(* LS Electric XG5000 project: XMC_E16A_ModTCP_Client *)
(* PLC LSPLC *)
(* module base 0 slot 0: Input/Output Module:XMC-DN24 (DC 24V Input 8Points/TR output 16Points) *)
(* module base 0 slot 1: Internal Analog Input/Output:XMF-AH04E (A/D voltage/current 2 channels, D/A voltage 2 channels) *)
(* task Periodic Task: Kind=2 *)
(* task Initialization Task: Kind=1 *)
(* task NC Program: Kind=6 *)

PROGRAM ModTCP_Read_FBs (* task: Scan Program *)
(* program showing examples of reading data from a Mod TCP server *)
VAR
    doFC1 : BOOL;
    doFC2 : BOOL;
    doFC3 : BOOL;
    doFC4 : BOOL; (* run function code 4 fb *)
    ErrorCount : INT;
    FC1 : MODBUS_READ_COILS_FC01; (* function code 1 fb *)
    fc1Data : ARRAY[0..1999] OF BOOL;
    FC1_UnitID : USINT; (* UnitID for FC1 fb *)
    FC2 : MODBUS_READ_DISCRETE_INPUTS_FC02; (* function code 2 fb *)
    fc2Data : ARRAY[0..1999] OF BOOL;
    FC2_UnitID : USINT; (* UnitID for FC2 fb *)
    FC3 : MODBUS_READ_HOLDING_REGISTER_FC03; (* function code 3 fb *)
    fc3Data : ARRAY[0..124] OF UINT;
    FC3_UnitID : USINT; (* UnitID for FC3 fb *)
    FC4 : MODBUS_READ_INPUT_REGISTERS_FC04; (* function code 4 fb *)
    fc4Data : ARRAY[0..124] OF UINT; (* data for function code 4 *)
    FC4_UnitID : USINT; (* UnitID for FC4 fb *)
    ipAddr : ARRAY[0..3] OF USINT;
    NonSocketError : BOOL;
    ResetDelay1 : TMR;
    ResetDelay2 : TMR;
    ResetDelay3 : TMR;
    SocketError : BOOL;
    StartResDelay1 : BOOL;
    StartResDelay2 : BOOL;
    STRFindIndex : INT;
    TCP_CheckSock1 : SOCKET_SVCINFO;
    TCP_CheckState1 : BOOL;
    TCP_Close1 : BOOL;
    TCP_Connect1 : BOOL;
    TCP_Sock1 : SOCKET_TCPCONNECT;
    TCP_SockClose : SOCKET_CLOSE;
END_VAR
VAR
    _p1 : BOOL;
END_VAR

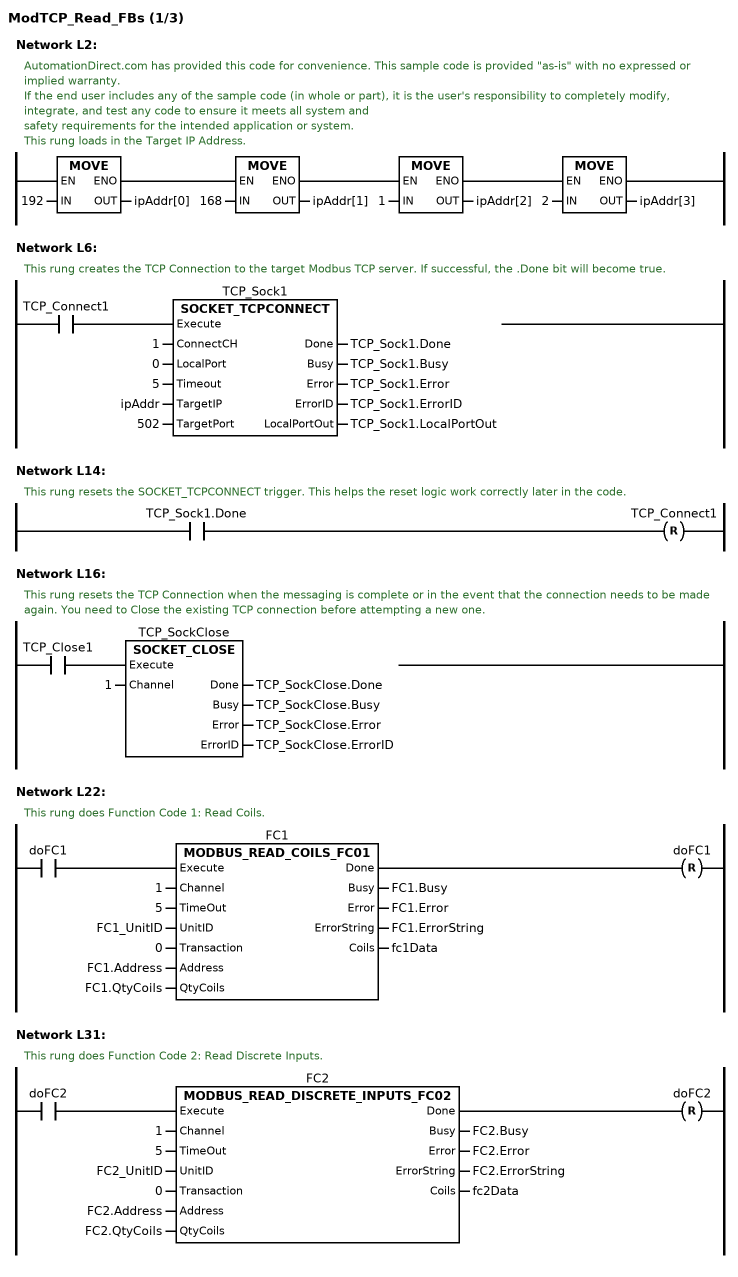
(* AutomationDirect.com has provided this code for convenience. This sample code is provided "as-is" with no expressed or implied warranty. / If the end user includes any of the sample code (in whole or part), it is the user's responsibility to completely modify, integrate, and test any code to ensure it meets all system and / safety requirements for the intended application or system. *)
(* This rung loads in the Target IP Address. *)
(* Rung L2 *)
ipAddr[0] := 192;
ipAddr[1] := 168;
ipAddr[2] := 1;
ipAddr[3] := 2;
(* This rung creates the TCP Connection to the target Modbus TCP server. If successful, the .Done bit will become true. *)
(* Rung L6 *)
TCP_Sock1(Execute := TCP_Connect1, ConnectCH := 1, LocalPort := 0, Timeout := 5, TargetIP := ipAddr, TargetPort := 502, Done => TCP_Sock1.Done, Busy => TCP_Sock1.Busy, Error => TCP_Sock1.Error, ErrorID => TCP_Sock1.ErrorID, LocalPortOut => TCP_Sock1.LocalPortOut);
(* This rung resets the SOCKET_TCPCONNECT trigger. This helps the reset logic work correctly later in the code. *)
(* Rung L14 *)
IF TCP_Sock1.Done THEN TCP_Connect1 := FALSE; END_IF;
(* This rung resets the TCP Connection when the messaging is complete or in the event that the connection needs to be made again. You need to Close the existing TCP connection before attempting a new one. *)
(* Rung L16 *)
TCP_SockClose(Execute := TCP_Close1, Channel := 1, Done => TCP_SockClose.Done, Busy => TCP_SockClose.Busy, Error => TCP_SockClose.Error, ErrorID => TCP_SockClose.ErrorID);
(* This rung does Function Code 1: Read Coils. *)
(* Rung L22 *)
FC1(Execute := doFC1, Channel := 1, TimeOut := 5, UnitID := FC1_UnitID, Transaction := 0, Address := FC1.Address, QtyCoils := FC1.QtyCoils, Busy => FC1.Busy, Error => FC1.Error, ErrorString => FC1.ErrorString, Coils => fc1Data);
IF FC1.Done THEN doFC1 := FALSE; END_IF;
(* This rung does Function Code 2: Read Discrete Inputs. *)
(* Rung L31 *)
FC2(Execute := doFC2, Channel := 1, TimeOut := 5, UnitID := FC2_UnitID, Transaction := 0, Address := FC2.Address, QtyCoils := FC2.QtyCoils, Busy => FC2.Busy, Error => FC2.Error, ErrorString => FC2.ErrorString, Coils => fc2Data);
IF FC2.Done THEN doFC2 := FALSE; END_IF;

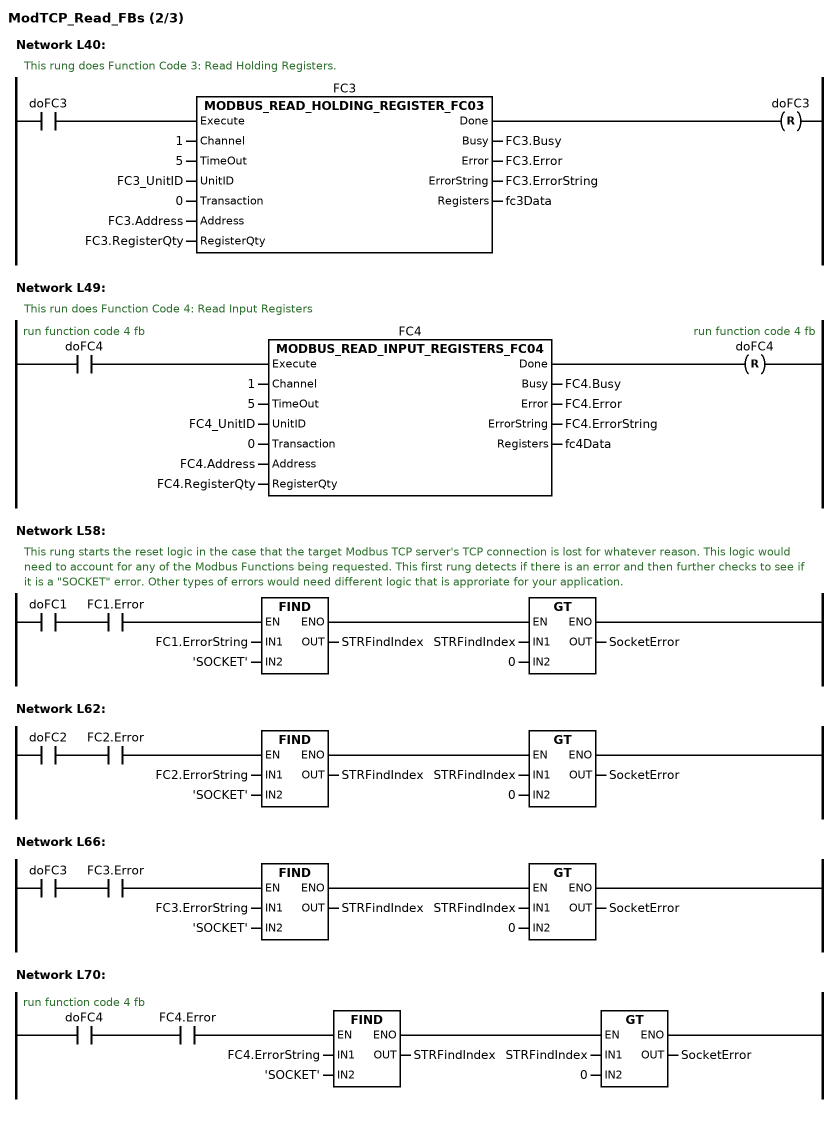
(* This rung does Function Code 3: Read Holding Registers. *)
(* Rung L40 *)
FC3(Execute := doFC3, Channel := 1, TimeOut := 5, UnitID := FC3_UnitID, Transaction := 0, Address := FC3.Address, RegisterQty := FC3.RegisterQty, Busy => FC3.Busy, Error => FC3.Error, ErrorString => FC3.ErrorString, Registers => fc3Data);
IF FC3.Done THEN doFC3 := FALSE; END_IF;
(* This run does Function Code 4: Read Input Registers *)
(* Rung L49 *)
FC4(Execute := doFC4, Channel := 1, TimeOut := 5, UnitID := FC4_UnitID, Transaction := 0, Address := FC4.Address, RegisterQty := FC4.RegisterQty, Busy => FC4.Busy, Error => FC4.Error, ErrorString => FC4.ErrorString, Registers => fc4Data);
IF FC4.Done THEN doFC4 := FALSE; END_IF;
(* This rung starts the reset logic in the case that the target Modbus TCP server's TCP connection is lost for whatever reason. This logic would need to account for any of the Modbus Functions being requested. This first rung detects if there is an error and then further checks to see if it is a "SOCKET" error. Other types of errors would need different logic that is approriate for your application. *)
(* Rung L58 *)
IF doFC1 AND FC1.Error THEN
    STRFindIndex := FIND(FC1.ErrorString, 'SOCKET');
    SocketError := STRFindIndex > 0;
END_IF;
(* Rung L62 *)
IF doFC2 AND FC2.Error THEN
    STRFindIndex := FIND(FC2.ErrorString, 'SOCKET');
    SocketError := STRFindIndex > 0;
END_IF;
(* Rung L66 *)
IF doFC3 AND FC3.Error THEN
    STRFindIndex := FIND(FC3.ErrorString, 'SOCKET');
    SocketError := STRFindIndex > 0;
END_IF;
(* Rung L70 *)
IF doFC4 AND FC4.Error THEN
    STRFindIndex := FIND(FC4.ErrorString, 'SOCKET');
    SocketError := STRFindIndex > 0;
END_IF;

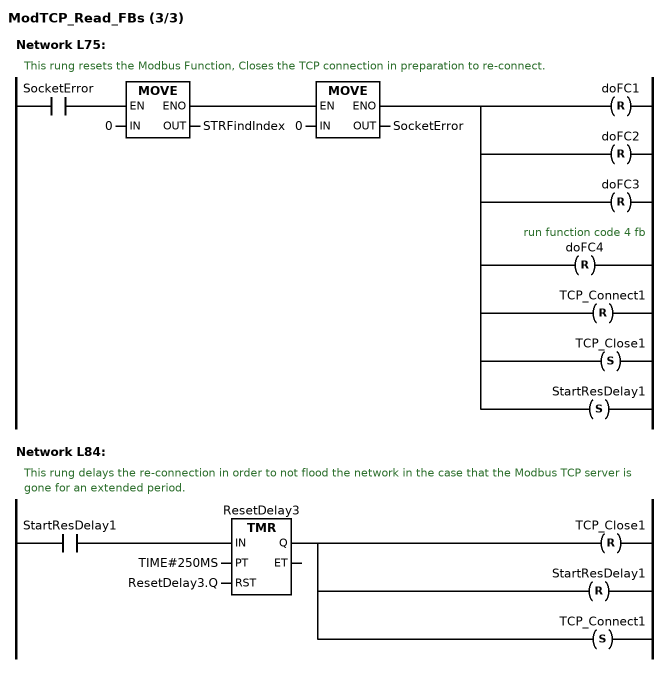
(* This rung resets the Modbus Function, Closes the TCP connection in preparation to re-connect. *)
(* Rung L75 *)
IF SocketError THEN STRFindIndex := 0; END_IF;
_p1 := SocketError;
IF _p1 THEN
    SocketError := 0;
    doFC1 := FALSE;
    doFC2 := FALSE;
    doFC3 := FALSE;
    doFC4 := FALSE;
    TCP_Connect1 := FALSE;
    TCP_Close1 := TRUE;
    StartResDelay1 := TRUE;
END_IF;
(* This rung delays the re-connection in order to not flood the network in the case that the Modbus TCP server is gone for an extended period. *)
(* Rung L84 *)
ResetDelay3(IN := StartResDelay1, PT := TIME#250MS, RST := ResetDelay3.Q);
IF ResetDelay3.Q THEN
    TCP_Close1 := FALSE;
    StartResDelay1 := FALSE;
    TCP_Connect1 := TRUE;
END_IF;
END_PROGRAM

PROGRAM ModTCP_Write_FBs (* task: Scan Program *)
(* example of ModBus TCP Write function blocks *)
VAR
    doFC15 : BOOL; (* execute function code 15 *)
    doFC16 : BOOL; (* execute function code 16 *)
    doFC5 : BOOL; (* execute function code 5 fb *)
    doFC6 : BOOL; (* execute function code 6 *)
    FC15 : MODBUS_WRITE_MULTIPLE_COILS_FC15; (* fb for function code 15 *)
    FC15_data : ARRAY[0..1967] OF BOOL;
    FC15_UnitID : USINT;
    FC16 : MODBUS_WRITE_MULTIPLE_REGISTERS_FC16; (* fb for function code 16 *)
    FC16_data : ARRAY[0..122] OF UINT;
    FC16_UnitID : USINT;
    FC5 : MODBUS_WRITE_SINGLE_COIL_FC05; (* function code 5 fb *)
    FC5_data : BOOL; (* data for fc5 *)
    FC5_UnitID : USINT;
    FC6 : MODBUS_WRITE_SINGLE_REGISTER_FC06; (* fb for function code 6 *)
    FC6_data : UINT;
    FC6_UnitID : USINT;
    ipAddr : ARRAY[0..3] OF USINT;
    ResetDelay3 : TMR;
    SocketError : BOOL;
    StartResDelay1 : BOOL;
    STRFindIndex : INT;
    TCP_Close1 : BOOL;
    TCP_Connect1 : BOOL;
    TCP_Sock1 : SOCKET_TCPCONNECT;
    TCP_SockClose : SOCKET_CLOSE;
END_VAR
VAR
    _p1 : BOOL;
END_VAR

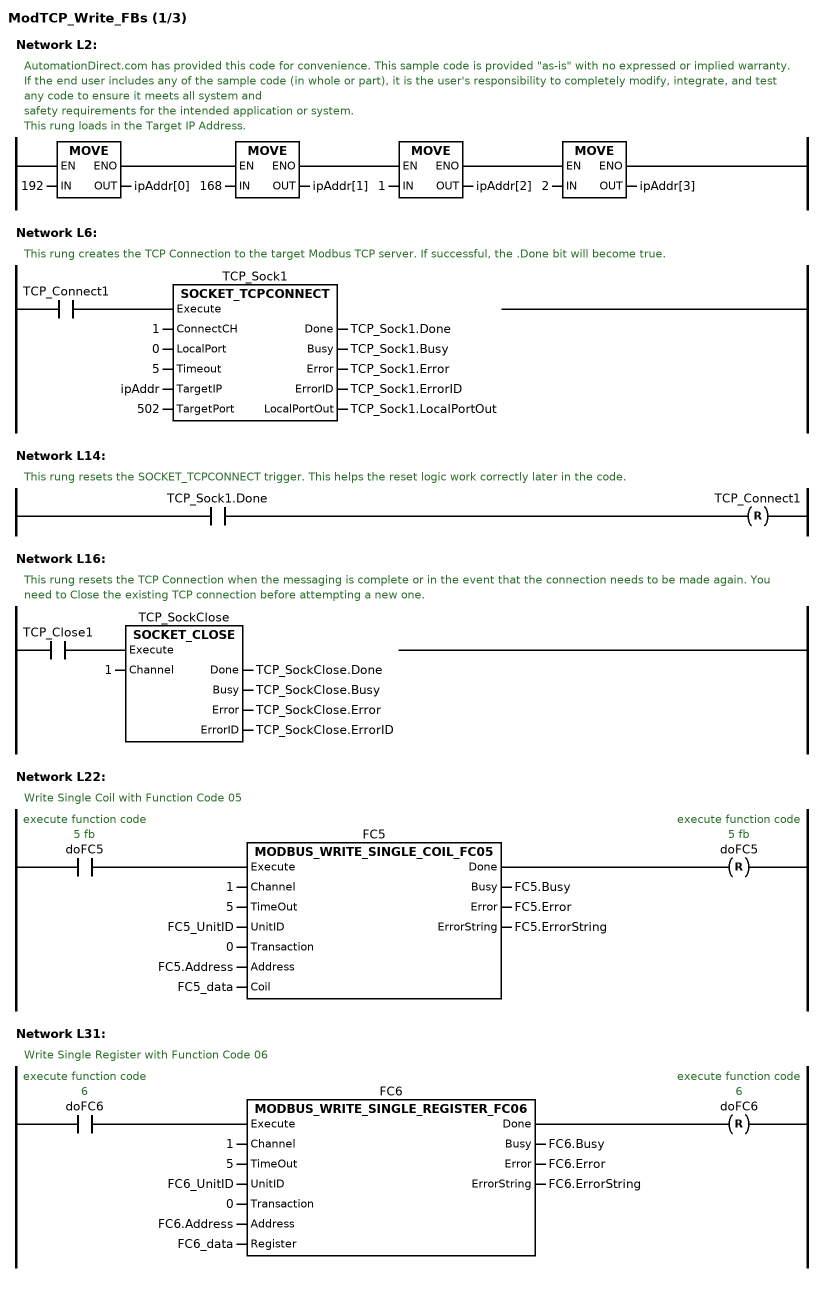
(* AutomationDirect.com has provided this code for convenience. This sample code is provided "as-is" with no expressed or implied warranty. / If the end user includes any of the sample code (in whole or part), it is the user's responsibility to completely modify, integrate, and test any code to ensure it meets all system and / safety requirements for the intended application or system. *)
(* This rung loads in the Target IP Address. *)
(* Rung L2 *)
ipAddr[0] := 192;
ipAddr[1] := 168;
ipAddr[2] := 1;
ipAddr[3] := 2;
(* This rung creates the TCP Connection to the target Modbus TCP server. If successful, the .Done bit will become true. *)
(* Rung L6 *)
TCP_Sock1(Execute := TCP_Connect1, ConnectCH := 1, LocalPort := 0, Timeout := 5, TargetIP := ipAddr, TargetPort := 502, Done => TCP_Sock1.Done, Busy => TCP_Sock1.Busy, Error => TCP_Sock1.Error, ErrorID => TCP_Sock1.ErrorID, LocalPortOut => TCP_Sock1.LocalPortOut);
(* This rung resets the SOCKET_TCPCONNECT trigger. This helps the reset logic work correctly later in the code. *)
(* Rung L14 *)
IF TCP_Sock1.Done THEN TCP_Connect1 := FALSE; END_IF;
(* This rung resets the TCP Connection when the messaging is complete or in the event that the connection needs to be made again. You need to Close the existing TCP connection before attempting a new one. *)
(* Rung L16 *)
TCP_SockClose(Execute := TCP_Close1, Channel := 1, Done => TCP_SockClose.Done, Busy => TCP_SockClose.Busy, Error => TCP_SockClose.Error, ErrorID => TCP_SockClose.ErrorID);
(* Write Single Coil with Function Code 05 *)
(* Rung L22 *)
FC5(Execute := doFC5, Channel := 1, TimeOut := 5, UnitID := FC5_UnitID, Transaction := 0, Address := FC5.Address, Coil := FC5_data, Busy => FC5.Busy, Error => FC5.Error, ErrorString => FC5.ErrorString);
IF FC5.Done THEN doFC5 := FALSE; END_IF;
(* Write Single Register with Function Code 06 *)
(* Rung L31 *)
FC6(Execute := doFC6, Channel := 1, TimeOut := 5, UnitID := FC6_UnitID, Transaction := 0, Address := FC6.Address, Register := FC6_data, Busy => FC6.Busy, Error => FC6.Error, ErrorString => FC6.ErrorString);
IF FC6.Done THEN doFC6 := FALSE; END_IF;

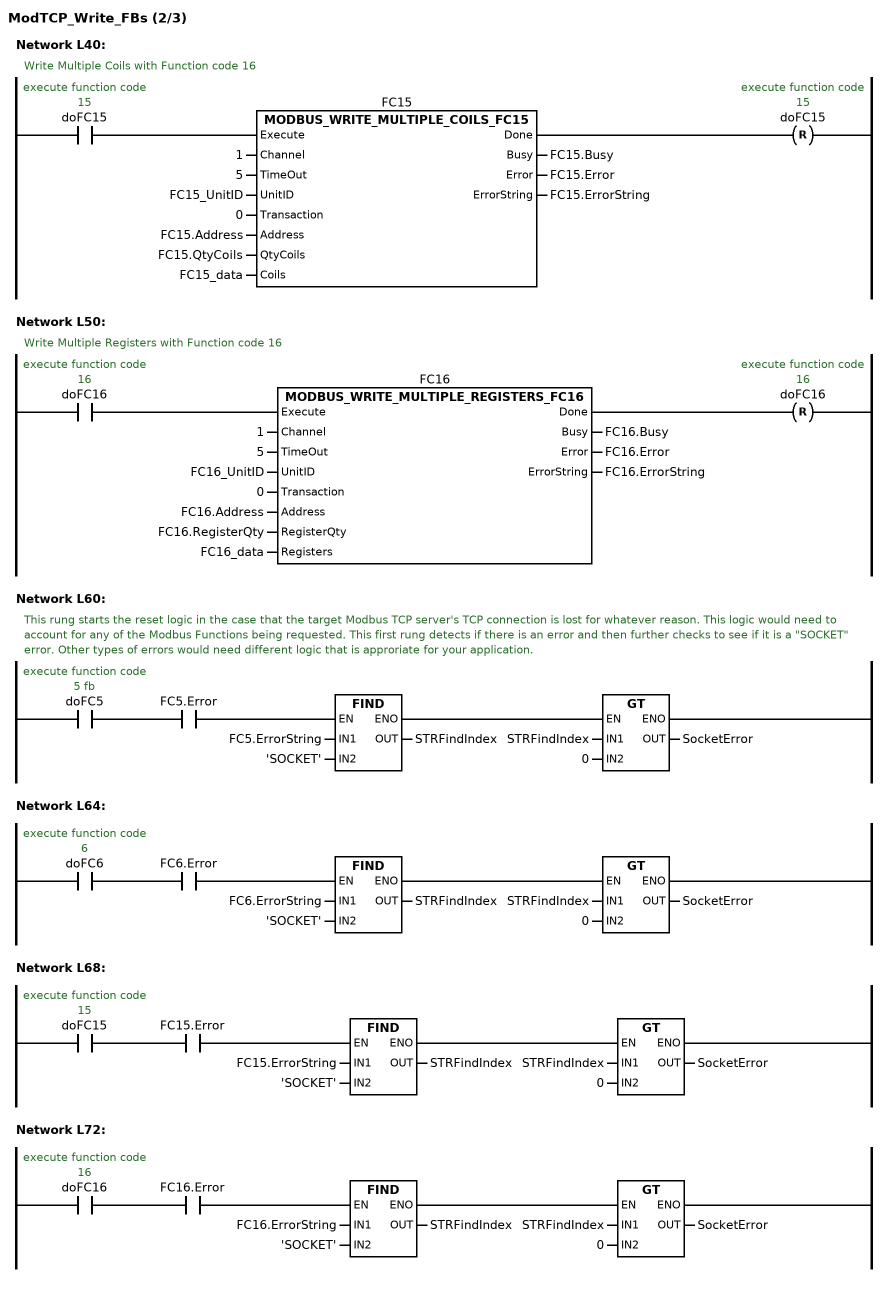
(* Write Multiple Coils with Function code 16 *)
(* Rung L40 *)
FC15(Execute := doFC15, Channel := 1, TimeOut := 5, UnitID := FC15_UnitID, Transaction := 0, Address := FC15.Address, QtyCoils := FC15.QtyCoils, Coils := FC15_data, Busy => FC15.Busy, Error => FC15.Error, ErrorString => FC15.ErrorString);
IF FC15.Done THEN doFC15 := FALSE; END_IF;
(* Write Multiple Registers with Function code 16 *)
(* Rung L50 *)
FC16(Execute := doFC16, Channel := 1, TimeOut := 5, UnitID := FC16_UnitID, Transaction := 0, Address := FC16.Address, RegisterQty := FC16.RegisterQty, Registers := FC16_data, Busy => FC16.Busy, Error => FC16.Error, ErrorString => FC16.ErrorString);
IF FC16.Done THEN doFC16 := FALSE; END_IF;
(* This rung starts the reset logic in the case that the target Modbus TCP server's TCP connection is lost for whatever reason. This logic would need to account for any of the Modbus Functions being requested. This first rung detects if there is an error and then further checks to see if it is a "SOCKET" error. Other types of errors would need different logic that is approriate for your application. *)
(* Rung L60 *)
IF doFC5 AND FC5.Error THEN
    STRFindIndex := FIND(FC5.ErrorString, 'SOCKET');
    SocketError := STRFindIndex > 0;
END_IF;
(* Rung L64 *)
IF doFC6 AND FC6.Error THEN
    STRFindIndex := FIND(FC6.ErrorString, 'SOCKET');
    SocketError := STRFindIndex > 0;
END_IF;
(* Rung L68 *)
IF doFC15 AND FC15.Error THEN
    STRFindIndex := FIND(FC15.ErrorString, 'SOCKET');
    SocketError := STRFindIndex > 0;
END_IF;
(* Rung L72 *)
IF doFC16 AND FC16.Error THEN
    STRFindIndex := FIND(FC16.ErrorString, 'SOCKET');
    SocketError := STRFindIndex > 0;
END_IF;

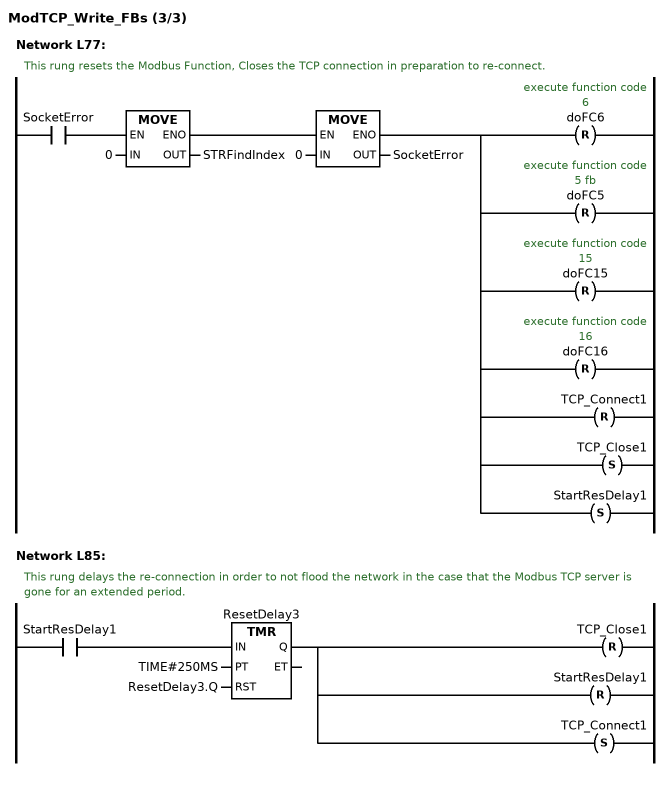
(* This rung resets the Modbus Function, Closes the TCP connection in preparation to re-connect. *)
(* Rung L77 *)
IF SocketError THEN STRFindIndex := 0; END_IF;
_p1 := SocketError;
IF _p1 THEN
    SocketError := 0;
    doFC6 := FALSE;
    doFC5 := FALSE;
    doFC15 := FALSE;
    doFC16 := FALSE;
    TCP_Connect1 := FALSE;
    TCP_Close1 := TRUE;
    StartResDelay1 := TRUE;
END_IF;
(* This rung delays the re-connection in order to not flood the network in the case that the Modbus TCP server is gone for an extended period. *)
(* Rung L85 *)
ResetDelay3(IN := StartResDelay1, PT := TIME#250MS, RST := ResetDelay3.Q);
IF ResetDelay3.Q THEN
    TCP_Close1 := FALSE;
    StartResDelay1 := FALSE;
    TCP_Connect1 := TRUE;
END_IF;
END_PROGRAM